// TwinCAT 3 PLC project PLC
// ProgramVersion: 3.1.4023.0
// libraries:
//   Tc2_Standard, * (Beckhoff Automation GmbH)
//   Tc2_System, * (Beckhoff Automation GmbH)
//   Tc3_Module, * (Beckhoff Automation GmbH)
// project tree:
//   CreateIndirectBinding/ PRG_IndirectBinding.TcPOU
//   DUT/ E_Pump_State.TcDUT, ST_Pump.TcDUT
//   / PlcTask.TcTTO
// real-time tasks:
//   TASK PlcTask: cycle T#10ms, priority 20, ADS port 350

CONFIGURATION PLC
    RESOURCE PLC ON TwinCAT3
        TASK PlcTask(INTERVAL := T#10ms, PRIORITY := 20);
        PROGRAM PRG_IndirectBinding WITH PlcTask : PRG_IndirectBinding;
    END_RESOURCE
END_CONFIGURATION

// ---- DUT/E_Pump_State.TcDUT
{attribute 'qualified_only'}
{attribute 'strict'}
TYPE E_Pump_State :
(
	Stopped := 0,
	Starting,
	Runing,
	Error
);
END_TYPE

// ---- DUT/ST_Pump.TcDUT
TYPE ST_Pump :
STRUCT
    Name 			: STRING;
	Speed			: LREAL;
	State			: E_Pump_State;
	Start			: BOOL;
	Stop			: BOOL;
END_STRUCT
END_TYPE

// ---- CreateIndirectBinding/PRG_IndirectBinding.TcPOU
PROGRAM PRG_IndirectBinding
VAR
	xInit			:BOOL:=TRUE;
	arString		:ARRAY[0..Upper] OF STRING;
	Pumps			:ARRAY[0..Upper] OF ST_Pump;	
END_VAR
VAR CONSTANT
	Upper			:UINT:=3;
END_VAR
VAR_TEMP
	i				:UDINT;
END_VAR

IF xInit THEN
	xInit		:=FALSE;
	FOR i:=0 TO Upper DO
		arString[i]		:=CONCAT('This is Index:',TO_STRING(i));
		Pumps[i].Name	:=CONCAT('Pump ', TO_STRING(i));
		Pumps[i].State  := E_Pump_State.Runing;		
	END_FOR
END_IF

FOR i:=0 TO Upper DO
	Pumps[i].Speed	:=Pumps[i].Speed+(i+1);
END_FOR

END_PROGRAM
